// TIA Portal V18 export
DATA_BLOCK "Heater_Control_DB"   // DB37
VERSION : 0.1
// stored: AutoNumber true, DBAccessibleFromOPCUA true, InstanceOfName IR_Heater_Control, InstanceOfType FB
"IR_Heater_Control"
   // VAR_INPUT
   //    MachineNumber : Int;
   //    Mode : Int;
   //    DoorSenor : Bool;
   //    RollerON { ExternalAccessible := 'False'; ExternalVisible := 'False'; ExternalWritable := 'False'} : Bool;
   //    Heater_Safety_PDL { ExternalAccessible := 'False'; ExternalVisible := 'False'; ExternalWritable := 'False'} : Real;
   //    Heater_PWM_address { ExternalAccessible := 'False'; ExternalVisible := 'False'; ExternalWritable := 'False'} : HW_PWM;
   //    Heater_Setpoint { ExternalAccessible := 'False'; ExternalVisible := 'False'; ExternalWritable := 'False'} : Real;
   //    "E-STOP" { ExternalAccessible := 'False'; ExternalVisible := 'False'; ExternalWritable := 'False'} : Bool;
   //    Heater_ON_OFF { ExternalAccessible := 'False'; ExternalVisible := 'False'; ExternalWritable := 'False'} : Bool;
   //    FeedboxHeating : Bool;
   //    PrintboxHeating : Bool;
   //    AxisYActualPosition : DInt;
   //    AxisYActualVelocity : Real;
   //    FeedboxStartMachine : DInt;
   //    FeedboxEndMachine : DInt;
   //    PrintboxStartMachine : DInt;
   //    PrintboxEndMachine : DInt;
   //    HeaterTest : Bool;
   // END_VAR
   // VAR_OUTPUT
   //    Heater_Output : Bool;
   //    Heater_Pulse_Duration : Int;
   //    Heater_Error : Int;
   //    Heater_Output_Check : Int;
   //    RollerONWayBack : Bool;
   //    WrongPositionInput : Bool;
   // END_VAR
   // VAR
   //    Heater_Scale_LimitReductionBed : Real;
   //    Heater_Scale_LimitNoReduction : Real;
   //    Heater_Scale_Internal : Real;
   //    Heater_status : Bool;
   //    Heater_signal : Int;
   //    Heater_safety_input : Bool;
   //    Heater_error_code : Word;
   //    Heater_Output_Check_1 : Int;
   //    SafetyTime : Bool;
   //    ReverseDirectionPermission : Bool;
   //    ReverseDirection : Bool;
   //    HeaterStatusSave : Bool;
   //    HeaterStatusTimeExpired : Bool;
   //    TurningOnInAdvanceSTART : DInt;
   //    TurningOnInAdvanceEND : DInt;
   //    TurningOnInAdvanceRefresh : DInt;
   //    Position { ExternalAccessible := 'False'; ExternalVisible := 'False'; ExternalWritable := 'False'} : DInt;
   //    FeedboxHeatingON : Bool;
   //    PrintboxHeatingON : Bool;
   //    HeaterWayBack : Bool;
   //    MaintenanceSkipPositionPermission : Bool;
   //    MaintenanceSkipRoller : Bool;
   //    DevModeHeater : Bool;
   //    DevelopmentAddOn01 : Bool;
   // END_VAR
BEGIN
END_DATA_BLOCK
